PROGRAM Wash
VAR
	Blink_Timer: TP;
	Stop_Timer: TON;
	Memorize: BOOL;
END_VAR

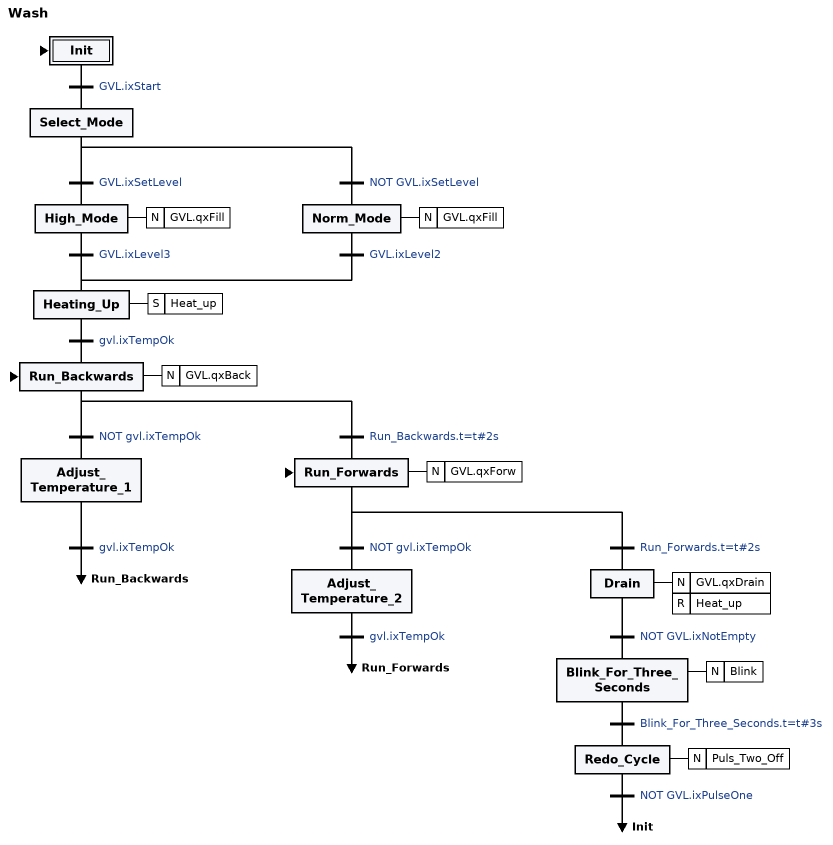
INITIAL_STEP Init:
END_STEP
TRANSITION FROM Init TO Select_Mode
    := GVL.ixStart;
END_TRANSITION
STEP Select_Mode:
END_STEP
TRANSITION FROM Select_Mode TO High_Mode
    := GVL.ixSetLevel;
END_TRANSITION
STEP High_Mode:
    GVL.qxFill(N);
END_STEP
TRANSITION FROM High_Mode TO Heating_Up
    := GVL.ixLevel3;
END_TRANSITION
TRANSITION FROM Select_Mode TO Norm_Mode
    := NOT GVL.ixSetLevel;
END_TRANSITION
STEP Norm_Mode:
    GVL.qxFill(N);
END_STEP
TRANSITION FROM Norm_Mode TO Heating_Up
    := GVL.ixLevel2;
END_TRANSITION
STEP Heating_Up:
    Heat_up(S);
END_STEP
TRANSITION FROM Heating_Up TO Run_Backwards
    := gvl.ixTempOk;
END_TRANSITION
STEP Run_Backwards:
    GVL.qxBack(N);
END_STEP
TRANSITION FROM Run_Backwards TO Adjust_Temperature_1
    := NOT gvl.ixTempOk;
END_TRANSITION
STEP Adjust_Temperature_1:
END_STEP
TRANSITION FROM Adjust_Temperature_1 TO Run_Backwards
    := gvl.ixTempOk;
END_TRANSITION
TRANSITION FROM Run_Backwards TO Run_Forwards
    := Run_Backwards.t=t#2s;
END_TRANSITION
STEP Run_Forwards:
    GVL.qxForw(N);
END_STEP
TRANSITION FROM Run_Forwards TO Adjust_Temperature_2
    := NOT gvl.ixTempOk;
END_TRANSITION
STEP Adjust_Temperature_2:
END_STEP
TRANSITION FROM Adjust_Temperature_2 TO Run_Forwards
    := gvl.ixTempOk;
END_TRANSITION
TRANSITION FROM Run_Forwards TO Drain
    := Run_Forwards.t=t#2s;
END_TRANSITION
STEP Drain:
    GVL.qxDrain(N);
    Heat_up(R);
END_STEP
TRANSITION FROM Drain TO Blink_For_Three_Seconds
    := NOT GVL.ixNotEmpty;
END_TRANSITION
STEP Blink_For_Three_Seconds:
    Blink(N);
END_STEP
TRANSITION FROM Blink_For_Three_Seconds TO Redo_Cycle
    := Blink_For_Three_Seconds.t=t#3s;
END_TRANSITION
STEP Redo_Cycle:
    Puls_Two_Off(N);
END_STEP
TRANSITION FROM Redo_Cycle TO Init
    := NOT GVL.ixPulseOne;
END_TRANSITION

ACTION Blink:
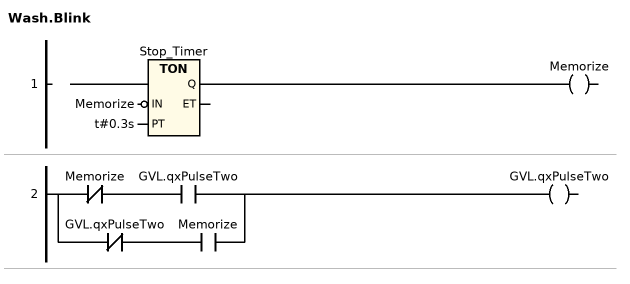
// NETWORK 1
Stop_Timer(IN := NOT Memorize, PT := t#0.3s); // TON
Memorize := Stop_Timer.Q;

// NETWORK 2
GVL.qxPulseTwo := NOT Memorize AND GVL.qxPulseTwo OR NOT GVL.qxPulseTwo AND Memorize;
END_ACTION

ACTION Heat_up:
IF gvl.iwCurrentTemp<=gvl.iwSetTemp THEN
	GVL.qxHeatingON := TRUE;
	
ELSE
	GVL.qxHeatingON := FALSE;
END_IF
END_ACTION

ACTION Puls_Two_Off:
gvl.qxPulseTwo:=FALSE;
END_ACTION

ACTION Reheat:

END_ACTION

END_PROGRAM

(* stored: Version 1.1.0.1, ProductVersion 3.1.4024.12
   POU Wash: Id {33924ad3-39a7-43fa-85a1-caf3c7fffb45}, SpecialFunc None
   Action Blink: Id {63eb1625-a8c8-40a4-a28b-23f4145206c8}
   Action Heat_up: Id {789ff41a-988b-4f9f-8bb2-4ac7fe978baf}
   Action Puls_Two_Off: Id {52161550-6f99-4287-a7cb-200499bbc840}
   Action Reheat: Id {7a1bfd87-c456-4e05-bf2a-6437d12ba39e} *)
